FUNCTION_BLOCK SELECT_5059E05E0748EACE (* Select *)
  (* Standard: 61499-2 *)
  (* Version 1.0, 22.10.2008, medusta, nxtControl GmbH, Initial Version *)
  PACKAGE UAO.Hackathon;
  (* Compiler Cpp *)
  {SET_ATTRIBUTE(Runtime.FBType.ImplementingType, Runtime.Standard#DYNGEN_MUX)}
  {SET_ATTRIBUTE(Configuration.GenericFBType.InterfaceParams, Runtime.Standard#CNT:=2;IN${CNT$}:STRING(255))}
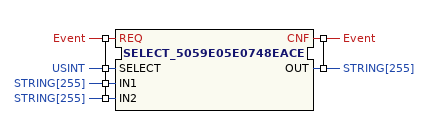
  EVENT_INPUT
    REQ WITH SELECT, IN1, IN2; (* Normal Execution Request *)
  END_EVENT
  EVENT_OUTPUT
    CNF WITH OUT; (* Execution Confirmation *)
  END_EVENT
  VAR_INPUT
    SELECT : USINT; (* Selector *)
    IN1 : STRING[255]; (* Argument *)
    IN2 : STRING[255]; (* Argument *)
  END_VAR
  VAR_OUTPUT
    OUT : STRING[255]; (* Result: IN1 or IN2 or ... according to the SELECT input (SELECT = 0 selects IN1) *)
  END_VAR
  EC_STATES
    START;
  END_STATES
END_FUNCTION_BLOCK
